FUNCTION_BLOCK FBlock (* Basic function block *)
  (* Standard: 61499 *)
  (* Version 1.0, 11/20/2015 9:00 AM, Kawsihen, Kawsihen_s Macintosh *)
  (* Compiler header: package mypackage *)
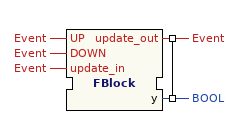
  EVENT_INPUT
    UP;
    DOWN;
    update_in;
  END_EVENT
  EVENT_OUTPUT
    update_out WITH y;
  END_EVENT
  VAR_OUTPUT
    y : BOOL;
  END_VAR
  VAR
    k : REAL;
    d : REAL;
    x : REAL;
    C1x : REAL;
  END_VAR
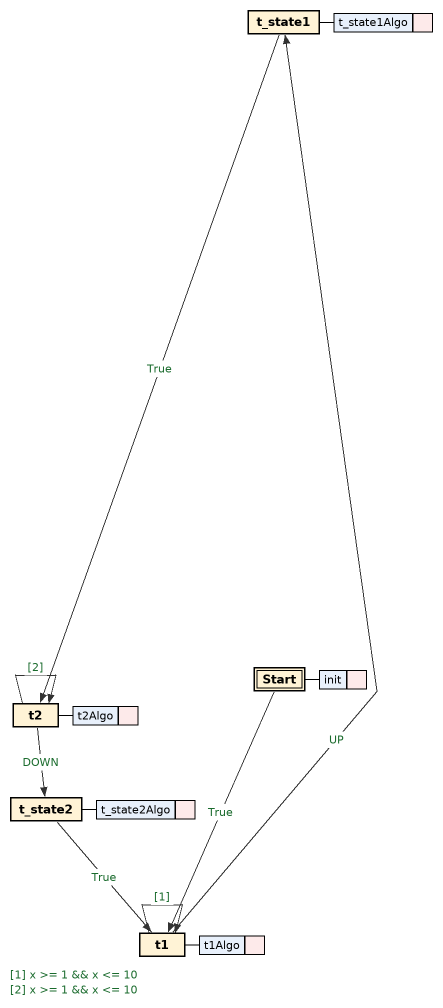
  EC_STATES
    Start : init;
    t1 : t1Algo;
    t2 : t2Algo;
    t_state1 : t_state1Algo;
    t_state2 : t_state2Algo;
  END_STATES
  EC_TRANSITIONS
    Start TO t1 := True;
    t1 TO t_state1 := UP;
    t_state1 TO t2 := True;
    t2 TO t_state2 := DOWN;
    t_state2 TO t1 := True;
    t1 TO t1 := x >= 1 && x <= 10;
    t2 TO t2 := x >= 1 && x <= 10;
  END_TRANSITIONS
  ALGORITHM t1Algo IN C:
me->C1x = 10.000;
me->x = (float) me->C1x*exp(-me->d*me->k/2);
me->k++;
  END_ALGORITHM
  ALGORITHM t2Algo IN C:
me->C1x = -10.000;
me->x = (float) me->C1x*exp(-me->d*me->k/2) + 11;
me->k++;
  END_ALGORITHM
  ALGORITHM init IN C:
me->d = 0.01;
me->k = 0;
;
  END_ALGORITHM
  ALGORITHM t_state1Algo IN C:
me->x = me->x;
me->k = 0;
  END_ALGORITHM
  ALGORITHM t_state2Algo IN C:
me->x = me->x;
me->k = 0;
  END_ALGORITHM
END_FUNCTION_BLOCK
